# EPICS autosave request: iocBoot/ioc1/dbSave/GS_Ah_.req
%
% BURT Request File
%
% $(P)GS:Ah:  Guard slits, Horizontal Aperture (type: Huber slits)
%

file assy.req ASSY=$(P)GS:Ah
$(P)GS:Ah:Invert
file mtr1.req MTR1=$(P)GS:mo
file mtr1.req MTR1=$(P)GS:mi
file drv1.req DRV1=$(P)GS:YO
file drv1.req DRV1=$(P)GS:YI
file axs1.req AXS1=$(P)GS:YC
file axs1.req AXS1=$(P)GS:YS
